// TIA Portal V17 export
// export: Created 2022-07-21T16:33:04.5420625Z, ExportSetting WithDefaults, WithReadOnly, DisplayName Totally Integrated Automation Portal, DisplayVersion V17, DisplayName TIA Portal Openness, DisplayVersion V17, DisplayName TIA Portal Version Control Interface, DisplayVersion V17, DisplayName SINAMICS Startdrive Advanced, DisplayVersion V17, DisplayName SINAMICS Startdrive G130, G150, S120, S150, SINAMICS MV, S210, DisplayVersion V17, DisplayName SINAMICS Startdrive G110M, G120, G120C, G120D, G120P, G115D, DisplayVersion V17, DisplayName STEP 7 Professional, DisplayVersion V17, DisplayName STEP 7 Safety, DisplayVersion V17, DisplayName WinCC Advanced, DisplayVersion V17
ScreenPopup "FRQ_002"  459x454
  ScreenLayer 
    FaceplateInstance "FRQ" at 1,1 size 458x453  FaceplateTypeName=IO@$@FRQ@$@FRQ V 3.0.40
      on ClosePoP: ShowPopupScreen(Name of the screen := , X coordinate := 0, Y coordinate := 0, Display mode := 0, Animation := -1, Animation speed := 1)
      CM_FRQ := FRQ_000
      Index := FRQ_Index
      Authorization := Operate
      Visibility := FRQ_FacePlateNo_Visible
      Item_number := CM_FRQ_Item_numbers
      Description_1 := CM_FRQ_description_1
